// Block: DEBUG_MES_Receive_Msg_Topic4XX

DATA_BLOCK DEBUG_MES_Receive_Msg_Topic4XX
VERSION : 0.1
   NON_RETAIN
   VAR
      DEBUG_RECEIVE : Struct
         Enable : Bool;
         AckChangeStep : Bool;
         ActualStep : Int;
      END_STRUCT;
      ACK_MSG_enable : Bool;
      NEW_MSG_401 : Struct
         ABILITA_FC : Bool;
         EXE_MSG : Bool;
         MSG : MES_Msg;
      END_STRUCT;
      NEW_MSG_402 : Struct
         ABILITA_FC : Bool;
         EXE_MSG : Bool;
         MSG : MES_Msg;
      END_STRUCT;
      NEW_MSG_403 : Struct
         ABILITA_FC : Bool;
         EXE_MSG : Bool;
         MSG : MES_Msg;
      END_STRUCT;
      NEW_MSG_410 : Struct
         ABILITA_FC : Bool;
         EXE_MSG : Bool;
         MSG : MES_Msg;
      END_STRUCT;
      NEW_MSG_412 : Struct
         ABILITA_FC : Bool;
         EXE_MSG : Bool;
         MSG : MES_Msg;
      END_STRUCT;
      NEW_MSG_422 : Struct
         ABILITA_FC : Bool;
         EXE_MSG : Bool;
         MSG : MES_Msg;
      END_STRUCT;
   END_VAR

BEGIN
   // No initialization required
END_DATA_BLOCK
